// TIA Portal V17 export
// export: Created 2024-09-02T12:50:27.3058177Z, ExportSetting WithDefaults, DisplayName Totally Integrated Automation Portal, DisplayVersion V17, DisplayName TIA Portal Openness, DisplayVersion V17, DisplayName TIA Portal Version Control Interface, DisplayVersion V17, DisplayName STEP 7 Professional, DisplayVersion V17, DisplayName STEP 7 Safety, DisplayVersion V17, DisplayName WinCC Professional, DisplayVersion V17
TYPE "TypeSKS_LIFT"
// stored: IsFailsafeCompliant false
   STRUCT
      "A" : Struct
         forward : Bool;
         middle : Bool;
         backward : Bool;
      END_STRUCT;
      H : Struct
         forward : Bool;
         middle : Bool;
         backward : Bool;
      END_STRUCT;
   END_STRUCT;
END_TYPE
